FUNCTION_BLOCK FB_CalcXRayDeltaMock EXTENDS FB_FalliblePublicMock IMPLEMENTS I_CalcXRayDelta
VAR
    fbResult : FB_QuantityLREALPublic(Units := '1');
END_VAR


METHOD Calculate
VAR_INPUT
    MaterialFormula : T_MaxString;
END_VAR
VAR_IN_OUT
    Delta : FB_QuantityLREALPublic(Units := '1');
END_VAR

Delta := fbResult;
END_METHOD


METHOD SetResult
VAR_INPUT
    Result : I_QuantityLREAL;
END_VAR

fbResult.Copy(QuantityToCopy := Result);
END_METHOD


METHOD SetValid

fbResult.Val := 1.0;
fbResult.Units := '1';
fbResult.ClearError();
ClearError();
END_METHOD

END_FUNCTION_BLOCK

(* stored: Version 1.1.0.1
   POU FB_CalcXRayDeltaMock: Id {7e76b36a-b6f5-47d3-8356-cf5207a967e6}, SpecialFunc None
   Method Calculate: Id {5bac6286-2214-4e59-adf7-609a7f98ff61}
   Method SetResult: Id {46e7158a-7ca6-4c4a-904d-ba67c1b04a23}
   Method SetValid: Id {e4af4d1f-4e6c-4927-9bea-b5784d00c67b} *)
